{attribute 'GeneratedUsingTerminal: EL3773-0000-0016'}
{attribute addProperty BoxType "EL3773-0000-0016"}
{attribute addProperty Id "I3_SAMPLESAT %I*I3_SAMPLES_2D13B74B20"}
{attribute addProperty CRC "363678031"}
{attribute addProperty Size "20"}
TYPE L3_Current_Samples_15AD494F EXTENDS InputBase_8311D824 :
STRUCT
	{attribute addProperty Name "I3_SAMPLES"}
	I3_SAMPLES AT %I* : I3_SAMPLES_2D13B74B;
END_STRUCT
END_TYPE

(* stored: Version 1.2.0.0, ProductVersion 3.1.4024.9
   DUT L3_Current_Samples_15AD494F: Id {417fcfae-666f-4348-b86f-c6b727cce64f} *)
